PROGRAM BasketBadCtrl
VAR
	ARfbStnBadAssignCtrl: ARRAY [1..iStnQty] OF fbAssignBadBstCtrl;
	ARfbArmBadAssignCtrl: ARRAY [1..iArmQty] OF fbAssignBadBstCtrl;
	bGeneralAssignBadBasket: BOOL;

END_VAR

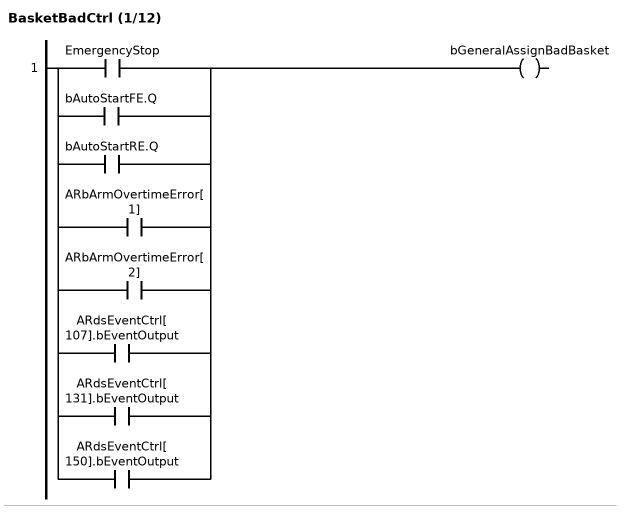
// NETWORK 1
bGeneralAssignBadBasket := EmergencyStop OR bAutoStartFE.Q OR bAutoStartRE.Q OR ARbArmOvertimeError[1] OR ARbArmOvertimeError[2] OR ARdsEventCtrl[107].bEventOutput OR ARdsEventCtrl[131].bEventOutput OR ARdsEventCtrl[150].bEventOutput;

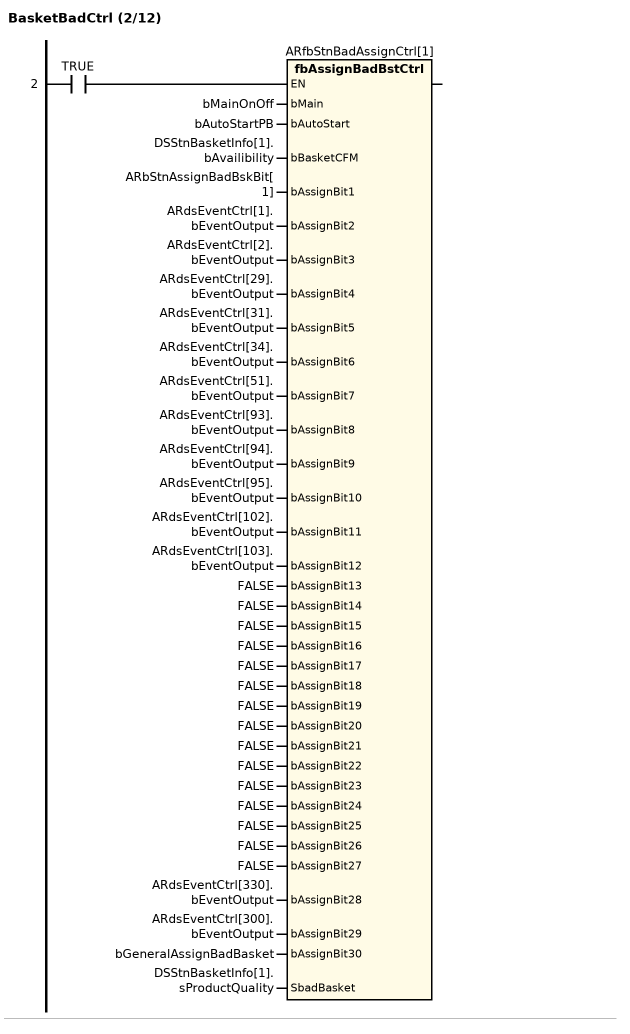
// NETWORK 2
ARfbStnBadAssignCtrl[1](
    bMain := bMainOnOff,
    bAutoStart := bAutoStartPB,
    bBasketCFM := DSStnBasketInfo[1].bAvailibility,
    bAssignBit1 := ARbStnAssignBadBskBit[1],
    bAssignBit2 := ARdsEventCtrl[1].bEventOutput,
    bAssignBit3 := ARdsEventCtrl[2].bEventOutput,
    bAssignBit4 := ARdsEventCtrl[29].bEventOutput,
    bAssignBit5 := ARdsEventCtrl[31].bEventOutput,
    bAssignBit6 := ARdsEventCtrl[34].bEventOutput,
    bAssignBit7 := ARdsEventCtrl[51].bEventOutput,
    bAssignBit8 := ARdsEventCtrl[93].bEventOutput,
    bAssignBit9 := ARdsEventCtrl[94].bEventOutput,
    bAssignBit10 := ARdsEventCtrl[95].bEventOutput,
    bAssignBit11 := ARdsEventCtrl[102].bEventOutput,
    bAssignBit12 := ARdsEventCtrl[103].bEventOutput,
    bAssignBit13 := FALSE,
    bAssignBit14 := FALSE,
    bAssignBit15 := FALSE,
    bAssignBit16 := FALSE,
    bAssignBit17 := FALSE,
    bAssignBit18 := FALSE,
    bAssignBit19 := FALSE,
    bAssignBit20 := FALSE,
    bAssignBit21 := FALSE,
    bAssignBit22 := FALSE,
    bAssignBit23 := FALSE,
    bAssignBit24 := FALSE,
    bAssignBit25 := FALSE,
    bAssignBit26 := FALSE,
    bAssignBit27 := FALSE,
    bAssignBit28 := ARdsEventCtrl[330].bEventOutput,
    bAssignBit29 := ARdsEventCtrl[300].bEventOutput,
    bAssignBit30 := bGeneralAssignBadBasket,
    SbadBasket := DSStnBasketInfo[1].sProductQuality); // fbAssignBadBstCtrl

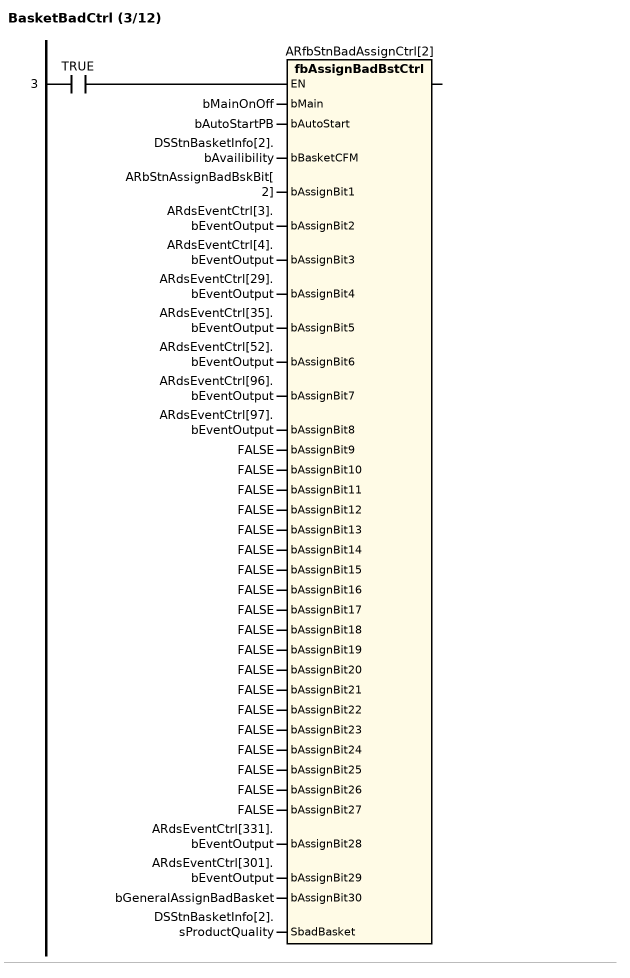
// NETWORK 3
ARfbStnBadAssignCtrl[2](
    bMain := bMainOnOff,
    bAutoStart := bAutoStartPB,
    bBasketCFM := DSStnBasketInfo[2].bAvailibility,
    bAssignBit1 := ARbStnAssignBadBskBit[2],
    bAssignBit2 := ARdsEventCtrl[3].bEventOutput,
    bAssignBit3 := ARdsEventCtrl[4].bEventOutput,
    bAssignBit4 := ARdsEventCtrl[29].bEventOutput,
    bAssignBit5 := ARdsEventCtrl[35].bEventOutput,
    bAssignBit6 := ARdsEventCtrl[52].bEventOutput,
    bAssignBit7 := ARdsEventCtrl[96].bEventOutput,
    bAssignBit8 := ARdsEventCtrl[97].bEventOutput,
    bAssignBit9 := FALSE,
    bAssignBit10 := FALSE,
    bAssignBit11 := FALSE,
    bAssignBit12 := FALSE,
    bAssignBit13 := FALSE,
    bAssignBit14 := FALSE,
    bAssignBit15 := FALSE,
    bAssignBit16 := FALSE,
    bAssignBit17 := FALSE,
    bAssignBit18 := FALSE,
    bAssignBit19 := FALSE,
    bAssignBit20 := FALSE,
    bAssignBit21 := FALSE,
    bAssignBit22 := FALSE,
    bAssignBit23 := FALSE,
    bAssignBit24 := FALSE,
    bAssignBit25 := FALSE,
    bAssignBit26 := FALSE,
    bAssignBit27 := FALSE,
    bAssignBit28 := ARdsEventCtrl[331].bEventOutput,
    bAssignBit29 := ARdsEventCtrl[301].bEventOutput,
    bAssignBit30 := bGeneralAssignBadBasket,
    SbadBasket := DSStnBasketInfo[2].sProductQuality); // fbAssignBadBstCtrl

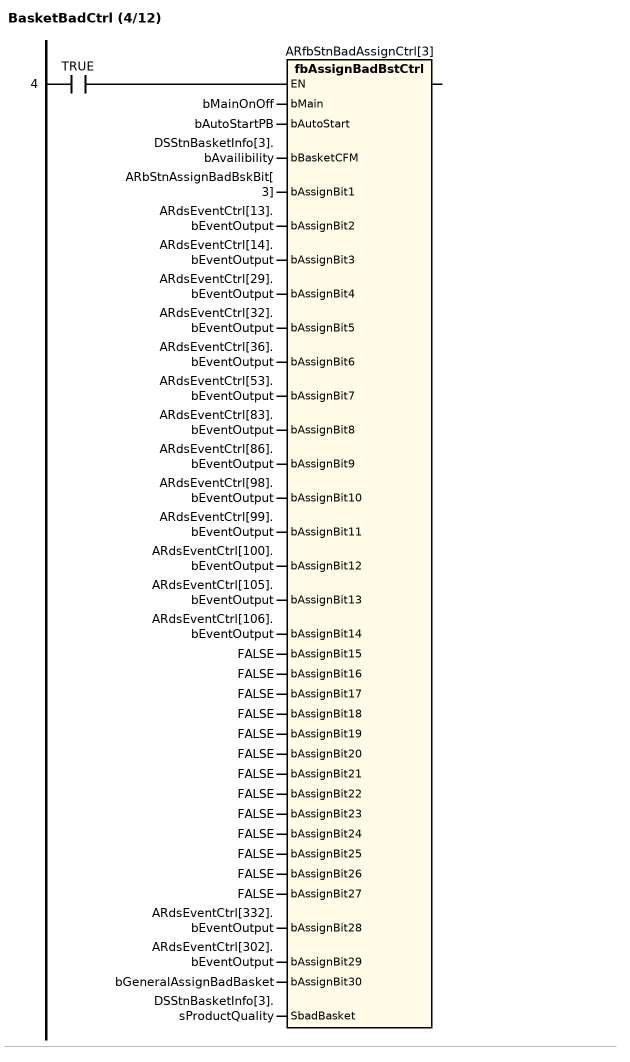
// NETWORK 4
ARfbStnBadAssignCtrl[3](
    bMain := bMainOnOff,
    bAutoStart := bAutoStartPB,
    bBasketCFM := DSStnBasketInfo[3].bAvailibility,
    bAssignBit1 := ARbStnAssignBadBskBit[3],
    bAssignBit2 := ARdsEventCtrl[13].bEventOutput,
    bAssignBit3 := ARdsEventCtrl[14].bEventOutput,
    bAssignBit4 := ARdsEventCtrl[29].bEventOutput,
    bAssignBit5 := ARdsEventCtrl[32].bEventOutput,
    bAssignBit6 := ARdsEventCtrl[36].bEventOutput,
    bAssignBit7 := ARdsEventCtrl[53].bEventOutput,
    bAssignBit8 := ARdsEventCtrl[83].bEventOutput,
    bAssignBit9 := ARdsEventCtrl[86].bEventOutput,
    bAssignBit10 := ARdsEventCtrl[98].bEventOutput,
    bAssignBit11 := ARdsEventCtrl[99].bEventOutput,
    bAssignBit12 := ARdsEventCtrl[100].bEventOutput,
    bAssignBit13 := ARdsEventCtrl[105].bEventOutput,
    bAssignBit14 := ARdsEventCtrl[106].bEventOutput,
    bAssignBit15 := FALSE,
    bAssignBit16 := FALSE,
    bAssignBit17 := FALSE,
    bAssignBit18 := FALSE,
    bAssignBit19 := FALSE,
    bAssignBit20 := FALSE,
    bAssignBit21 := FALSE,
    bAssignBit22 := FALSE,
    bAssignBit23 := FALSE,
    bAssignBit24 := FALSE,
    bAssignBit25 := FALSE,
    bAssignBit26 := FALSE,
    bAssignBit27 := FALSE,
    bAssignBit28 := ARdsEventCtrl[332].bEventOutput,
    bAssignBit29 := ARdsEventCtrl[302].bEventOutput,
    bAssignBit30 := bGeneralAssignBadBasket,
    SbadBasket := DSStnBasketInfo[3].sProductQuality); // fbAssignBadBstCtrl

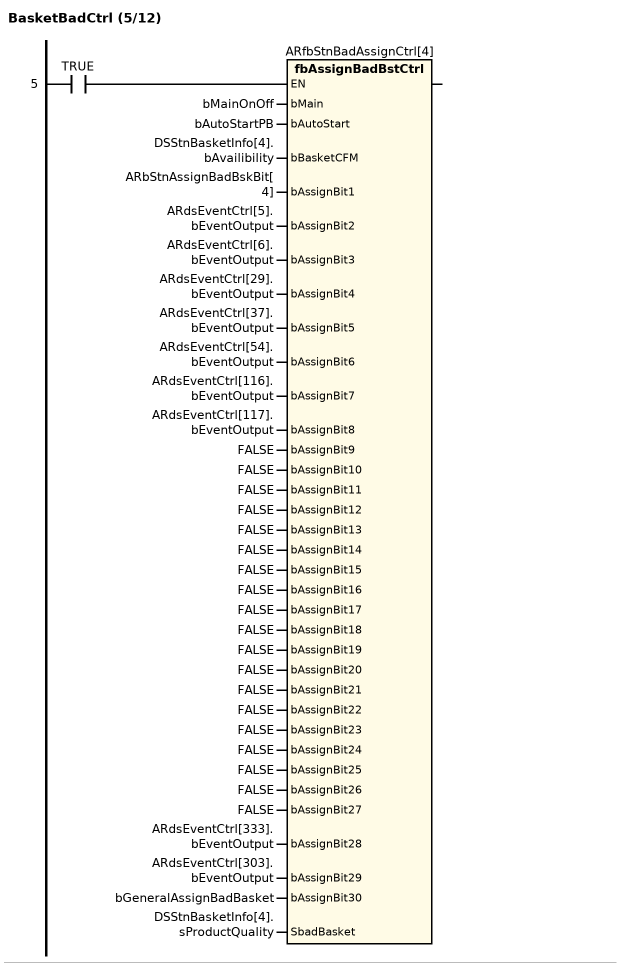
// NETWORK 5
ARfbStnBadAssignCtrl[4](
    bMain := bMainOnOff,
    bAutoStart := bAutoStartPB,
    bBasketCFM := DSStnBasketInfo[4].bAvailibility,
    bAssignBit1 := ARbStnAssignBadBskBit[4],
    bAssignBit2 := ARdsEventCtrl[5].bEventOutput,
    bAssignBit3 := ARdsEventCtrl[6].bEventOutput,
    bAssignBit4 := ARdsEventCtrl[29].bEventOutput,
    bAssignBit5 := ARdsEventCtrl[37].bEventOutput,
    bAssignBit6 := ARdsEventCtrl[54].bEventOutput,
    bAssignBit7 := ARdsEventCtrl[116].bEventOutput,
    bAssignBit8 := ARdsEventCtrl[117].bEventOutput,
    bAssignBit9 := FALSE,
    bAssignBit10 := FALSE,
    bAssignBit11 := FALSE,
    bAssignBit12 := FALSE,
    bAssignBit13 := FALSE,
    bAssignBit14 := FALSE,
    bAssignBit15 := FALSE,
    bAssignBit16 := FALSE,
    bAssignBit17 := FALSE,
    bAssignBit18 := FALSE,
    bAssignBit19 := FALSE,
    bAssignBit20 := FALSE,
    bAssignBit21 := FALSE,
    bAssignBit22 := FALSE,
    bAssignBit23 := FALSE,
    bAssignBit24 := FALSE,
    bAssignBit25 := FALSE,
    bAssignBit26 := FALSE,
    bAssignBit27 := FALSE,
    bAssignBit28 := ARdsEventCtrl[333].bEventOutput,
    bAssignBit29 := ARdsEventCtrl[303].bEventOutput,
    bAssignBit30 := bGeneralAssignBadBasket,
    SbadBasket := DSStnBasketInfo[4].sProductQuality); // fbAssignBadBstCtrl

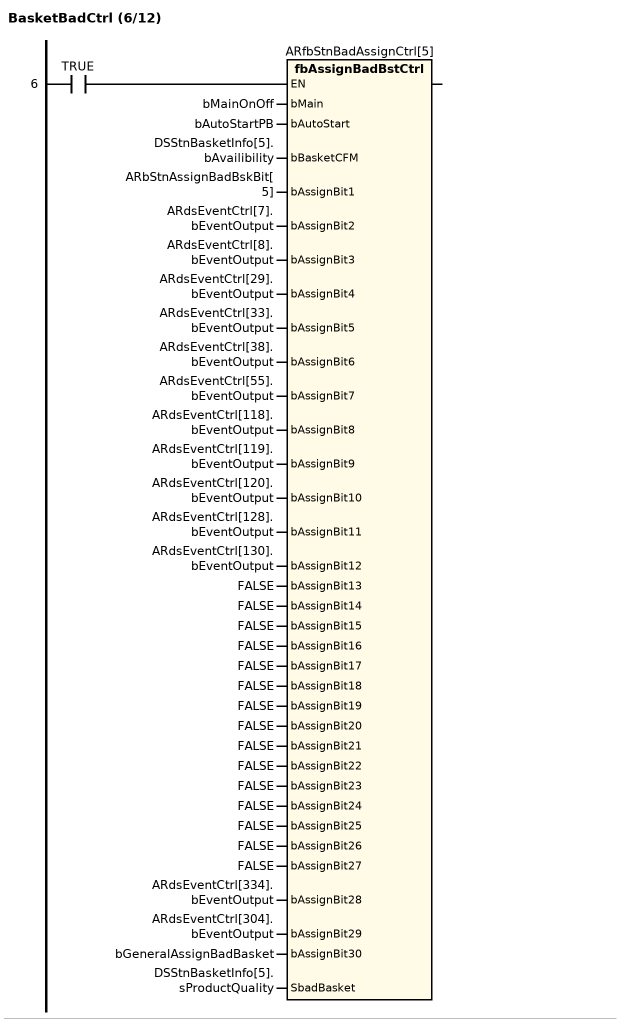
// NETWORK 6
ARfbStnBadAssignCtrl[5](
    bMain := bMainOnOff,
    bAutoStart := bAutoStartPB,
    bBasketCFM := DSStnBasketInfo[5].bAvailibility,
    bAssignBit1 := ARbStnAssignBadBskBit[5],
    bAssignBit2 := ARdsEventCtrl[7].bEventOutput,
    bAssignBit3 := ARdsEventCtrl[8].bEventOutput,
    bAssignBit4 := ARdsEventCtrl[29].bEventOutput,
    bAssignBit5 := ARdsEventCtrl[33].bEventOutput,
    bAssignBit6 := ARdsEventCtrl[38].bEventOutput,
    bAssignBit7 := ARdsEventCtrl[55].bEventOutput,
    bAssignBit8 := ARdsEventCtrl[118].bEventOutput,
    bAssignBit9 := ARdsEventCtrl[119].bEventOutput,
    bAssignBit10 := ARdsEventCtrl[120].bEventOutput,
    bAssignBit11 := ARdsEventCtrl[128].bEventOutput,
    bAssignBit12 := ARdsEventCtrl[130].bEventOutput,
    bAssignBit13 := FALSE,
    bAssignBit14 := FALSE,
    bAssignBit15 := FALSE,
    bAssignBit16 := FALSE,
    bAssignBit17 := FALSE,
    bAssignBit18 := FALSE,
    bAssignBit19 := FALSE,
    bAssignBit20 := FALSE,
    bAssignBit21 := FALSE,
    bAssignBit22 := FALSE,
    bAssignBit23 := FALSE,
    bAssignBit24 := FALSE,
    bAssignBit25 := FALSE,
    bAssignBit26 := FALSE,
    bAssignBit27 := FALSE,
    bAssignBit28 := ARdsEventCtrl[334].bEventOutput,
    bAssignBit29 := ARdsEventCtrl[304].bEventOutput,
    bAssignBit30 := bGeneralAssignBadBasket,
    SbadBasket := DSStnBasketInfo[5].sProductQuality); // fbAssignBadBstCtrl

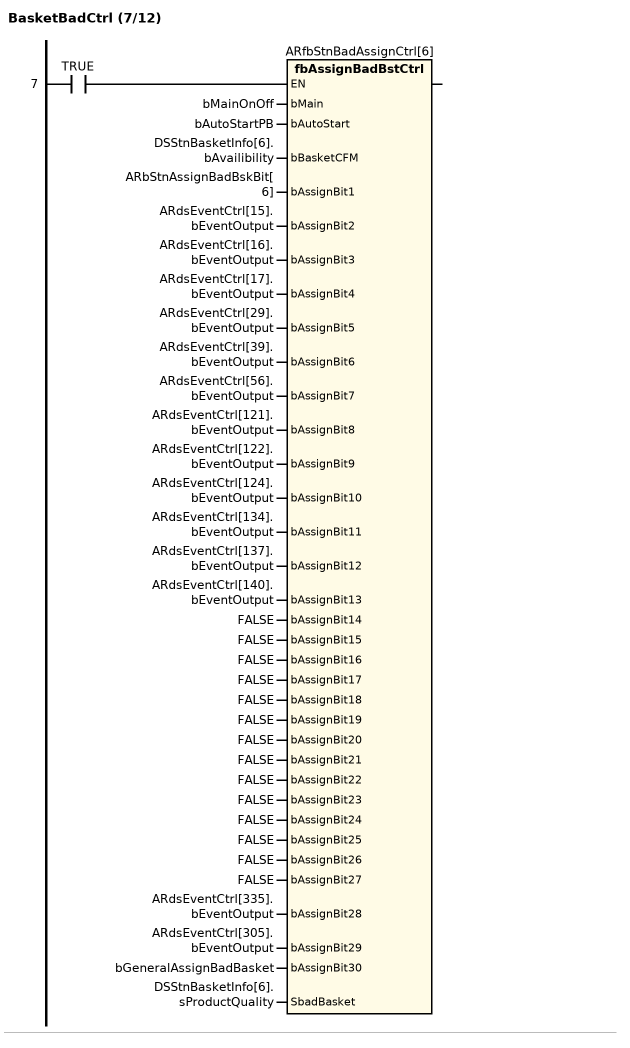
// NETWORK 7
ARfbStnBadAssignCtrl[6](
    bMain := bMainOnOff,
    bAutoStart := bAutoStartPB,
    bBasketCFM := DSStnBasketInfo[6].bAvailibility,
    bAssignBit1 := ARbStnAssignBadBskBit[6],
    bAssignBit2 := ARdsEventCtrl[15].bEventOutput,
    bAssignBit3 := ARdsEventCtrl[16].bEventOutput,
    bAssignBit4 := ARdsEventCtrl[17].bEventOutput,
    bAssignBit5 := ARdsEventCtrl[29].bEventOutput,
    bAssignBit6 := ARdsEventCtrl[39].bEventOutput,
    bAssignBit7 := ARdsEventCtrl[56].bEventOutput,
    bAssignBit8 := ARdsEventCtrl[121].bEventOutput,
    bAssignBit9 := ARdsEventCtrl[122].bEventOutput,
    bAssignBit10 := ARdsEventCtrl[124].bEventOutput,
    bAssignBit11 := ARdsEventCtrl[134].bEventOutput,
    bAssignBit12 := ARdsEventCtrl[137].bEventOutput,
    bAssignBit13 := ARdsEventCtrl[140].bEventOutput,
    bAssignBit14 := FALSE,
    bAssignBit15 := FALSE,
    bAssignBit16 := FALSE,
    bAssignBit17 := FALSE,
    bAssignBit18 := FALSE,
    bAssignBit19 := FALSE,
    bAssignBit20 := FALSE,
    bAssignBit21 := FALSE,
    bAssignBit22 := FALSE,
    bAssignBit23 := FALSE,
    bAssignBit24 := FALSE,
    bAssignBit25 := FALSE,
    bAssignBit26 := FALSE,
    bAssignBit27 := FALSE,
    bAssignBit28 := ARdsEventCtrl[335].bEventOutput,
    bAssignBit29 := ARdsEventCtrl[305].bEventOutput,
    bAssignBit30 := bGeneralAssignBadBasket,
    SbadBasket := DSStnBasketInfo[6].sProductQuality); // fbAssignBadBstCtrl

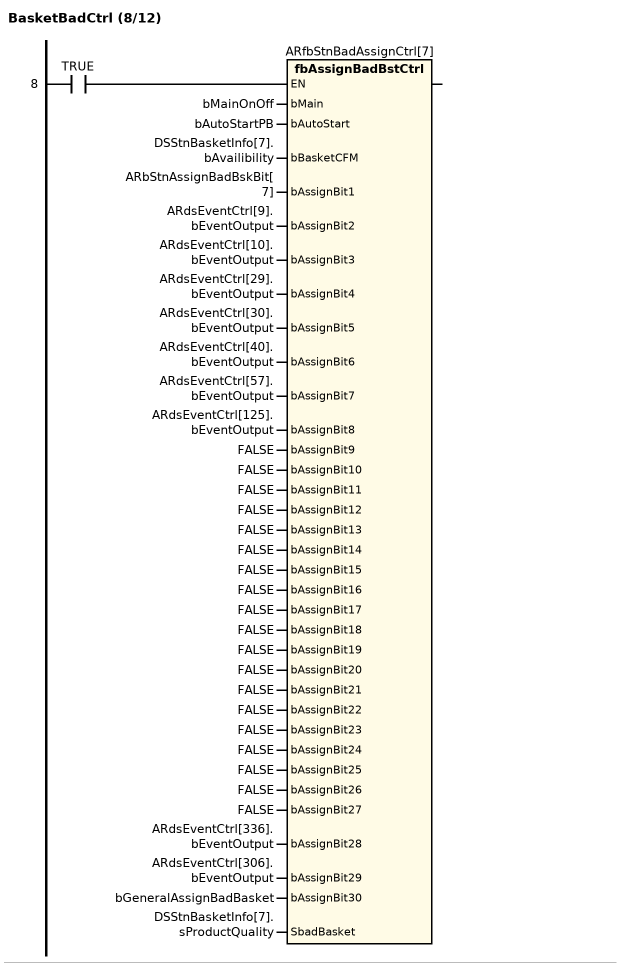
// NETWORK 8
ARfbStnBadAssignCtrl[7](
    bMain := bMainOnOff,
    bAutoStart := bAutoStartPB,
    bBasketCFM := DSStnBasketInfo[7].bAvailibility,
    bAssignBit1 := ARbStnAssignBadBskBit[7],
    bAssignBit2 := ARdsEventCtrl[9].bEventOutput,
    bAssignBit3 := ARdsEventCtrl[10].bEventOutput,
    bAssignBit4 := ARdsEventCtrl[29].bEventOutput,
    bAssignBit5 := ARdsEventCtrl[30].bEventOutput,
    bAssignBit6 := ARdsEventCtrl[40].bEventOutput,
    bAssignBit7 := ARdsEventCtrl[57].bEventOutput,
    bAssignBit8 := ARdsEventCtrl[125].bEventOutput,
    bAssignBit9 := FALSE,
    bAssignBit10 := FALSE,
    bAssignBit11 := FALSE,
    bAssignBit12 := FALSE,
    bAssignBit13 := FALSE,
    bAssignBit14 := FALSE,
    bAssignBit15 := FALSE,
    bAssignBit16 := FALSE,
    bAssignBit17 := FALSE,
    bAssignBit18 := FALSE,
    bAssignBit19 := FALSE,
    bAssignBit20 := FALSE,
    bAssignBit21 := FALSE,
    bAssignBit22 := FALSE,
    bAssignBit23 := FALSE,
    bAssignBit24 := FALSE,
    bAssignBit25 := FALSE,
    bAssignBit26 := FALSE,
    bAssignBit27 := FALSE,
    bAssignBit28 := ARdsEventCtrl[336].bEventOutput,
    bAssignBit29 := ARdsEventCtrl[306].bEventOutput,
    bAssignBit30 := bGeneralAssignBadBasket,
    SbadBasket := DSStnBasketInfo[7].sProductQuality); // fbAssignBadBstCtrl

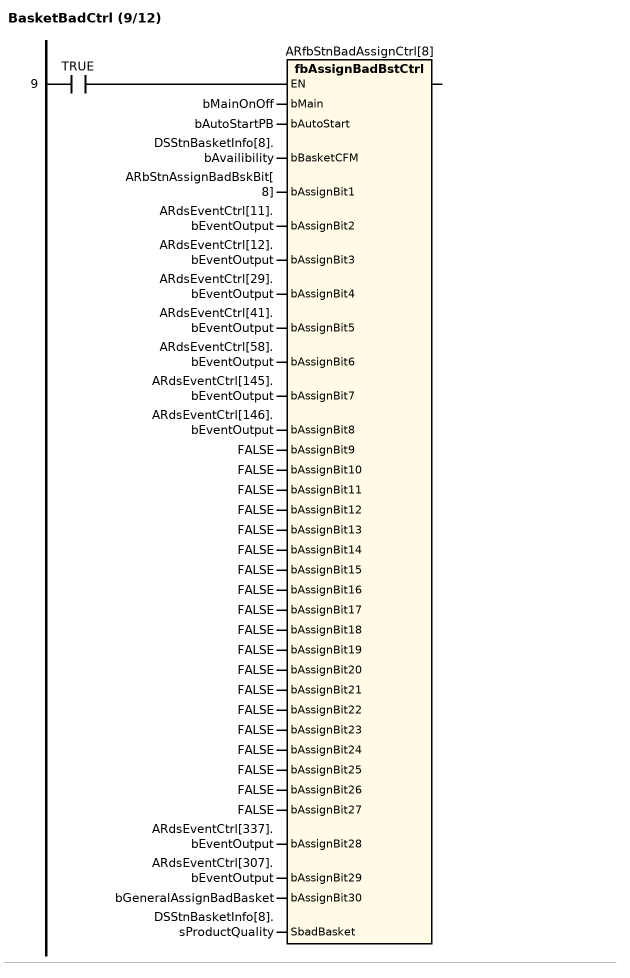
// NETWORK 9
ARfbStnBadAssignCtrl[8](
    bMain := bMainOnOff,
    bAutoStart := bAutoStartPB,
    bBasketCFM := DSStnBasketInfo[8].bAvailibility,
    bAssignBit1 := ARbStnAssignBadBskBit[8],
    bAssignBit2 := ARdsEventCtrl[11].bEventOutput,
    bAssignBit3 := ARdsEventCtrl[12].bEventOutput,
    bAssignBit4 := ARdsEventCtrl[29].bEventOutput,
    bAssignBit5 := ARdsEventCtrl[41].bEventOutput,
    bAssignBit6 := ARdsEventCtrl[58].bEventOutput,
    bAssignBit7 := ARdsEventCtrl[145].bEventOutput,
    bAssignBit8 := ARdsEventCtrl[146].bEventOutput,
    bAssignBit9 := FALSE,
    bAssignBit10 := FALSE,
    bAssignBit11 := FALSE,
    bAssignBit12 := FALSE,
    bAssignBit13 := FALSE,
    bAssignBit14 := FALSE,
    bAssignBit15 := FALSE,
    bAssignBit16 := FALSE,
    bAssignBit17 := FALSE,
    bAssignBit18 := FALSE,
    bAssignBit19 := FALSE,
    bAssignBit20 := FALSE,
    bAssignBit21 := FALSE,
    bAssignBit22 := FALSE,
    bAssignBit23 := FALSE,
    bAssignBit24 := FALSE,
    bAssignBit25 := FALSE,
    bAssignBit26 := FALSE,
    bAssignBit27 := FALSE,
    bAssignBit28 := ARdsEventCtrl[337].bEventOutput,
    bAssignBit29 := ARdsEventCtrl[307].bEventOutput,
    bAssignBit30 := bGeneralAssignBadBasket,
    SbadBasket := DSStnBasketInfo[8].sProductQuality); // fbAssignBadBstCtrl

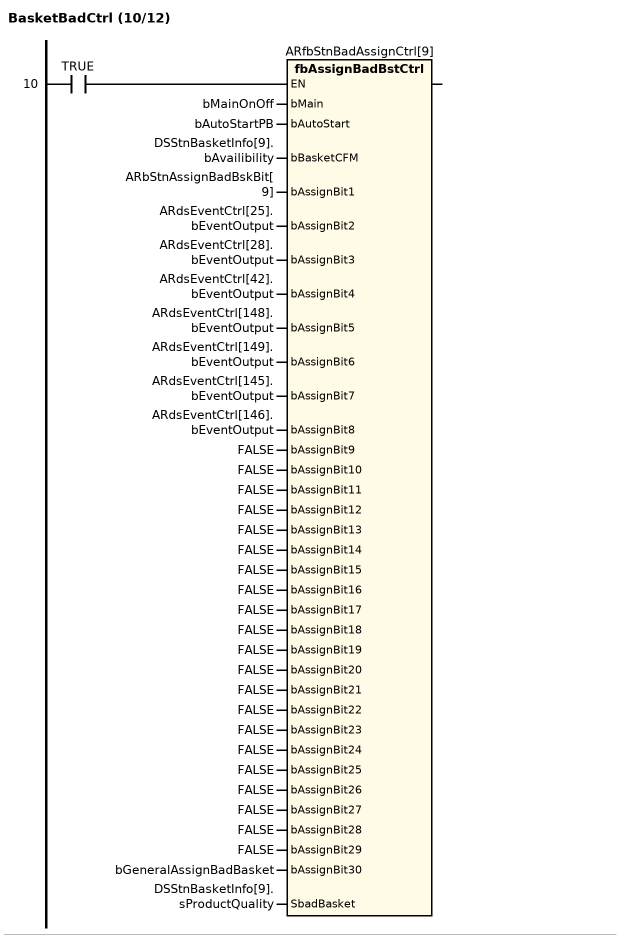
// NETWORK 10
ARfbStnBadAssignCtrl[9](
    bMain := bMainOnOff,
    bAutoStart := bAutoStartPB,
    bBasketCFM := DSStnBasketInfo[9].bAvailibility,
    bAssignBit1 := ARbStnAssignBadBskBit[9],
    bAssignBit2 := ARdsEventCtrl[25].bEventOutput,
    bAssignBit3 := ARdsEventCtrl[28].bEventOutput,
    bAssignBit4 := ARdsEventCtrl[42].bEventOutput,
    bAssignBit5 := ARdsEventCtrl[148].bEventOutput,
    bAssignBit6 := ARdsEventCtrl[149].bEventOutput,
    bAssignBit7 := ARdsEventCtrl[145].bEventOutput,
    bAssignBit8 := ARdsEventCtrl[146].bEventOutput,
    bAssignBit9 := FALSE,
    bAssignBit10 := FALSE,
    bAssignBit11 := FALSE,
    bAssignBit12 := FALSE,
    bAssignBit13 := FALSE,
    bAssignBit14 := FALSE,
    bAssignBit15 := FALSE,
    bAssignBit16 := FALSE,
    bAssignBit17 := FALSE,
    bAssignBit18 := FALSE,
    bAssignBit19 := FALSE,
    bAssignBit20 := FALSE,
    bAssignBit21 := FALSE,
    bAssignBit22 := FALSE,
    bAssignBit23 := FALSE,
    bAssignBit24 := FALSE,
    bAssignBit25 := FALSE,
    bAssignBit26 := FALSE,
    bAssignBit27 := FALSE,
    bAssignBit28 := FALSE,
    bAssignBit29 := FALSE,
    bAssignBit30 := bGeneralAssignBadBasket,
    SbadBasket := DSStnBasketInfo[9].sProductQuality); // fbAssignBadBstCtrl

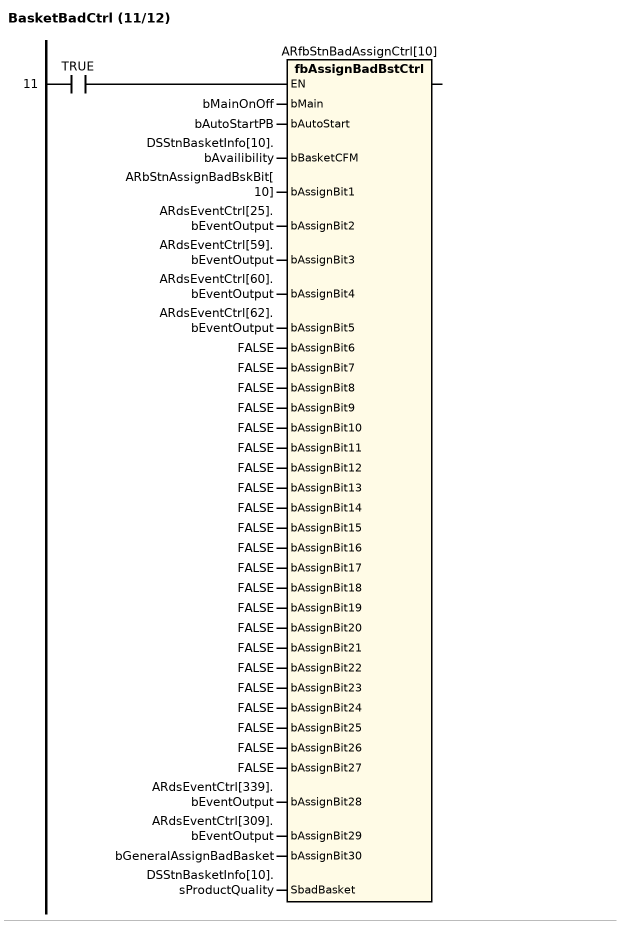
// NETWORK 11
ARfbStnBadAssignCtrl[10](
    bMain := bMainOnOff,
    bAutoStart := bAutoStartPB,
    bBasketCFM := DSStnBasketInfo[10].bAvailibility,
    bAssignBit1 := ARbStnAssignBadBskBit[10],
    bAssignBit2 := ARdsEventCtrl[25].bEventOutput,
    bAssignBit3 := ARdsEventCtrl[59].bEventOutput,
    bAssignBit4 := ARdsEventCtrl[60].bEventOutput,
    bAssignBit5 := ARdsEventCtrl[62].bEventOutput,
    bAssignBit6 := FALSE,
    bAssignBit7 := FALSE,
    bAssignBit8 := FALSE,
    bAssignBit9 := FALSE,
    bAssignBit10 := FALSE,
    bAssignBit11 := FALSE,
    bAssignBit12 := FALSE,
    bAssignBit13 := FALSE,
    bAssignBit14 := FALSE,
    bAssignBit15 := FALSE,
    bAssignBit16 := FALSE,
    bAssignBit17 := FALSE,
    bAssignBit18 := FALSE,
    bAssignBit19 := FALSE,
    bAssignBit20 := FALSE,
    bAssignBit21 := FALSE,
    bAssignBit22 := FALSE,
    bAssignBit23 := FALSE,
    bAssignBit24 := FALSE,
    bAssignBit25 := FALSE,
    bAssignBit26 := FALSE,
    bAssignBit27 := FALSE,
    bAssignBit28 := ARdsEventCtrl[339].bEventOutput,
    bAssignBit29 := ARdsEventCtrl[309].bEventOutput,
    bAssignBit30 := bGeneralAssignBadBasket,
    SbadBasket := DSStnBasketInfo[10].sProductQuality); // fbAssignBadBstCtrl

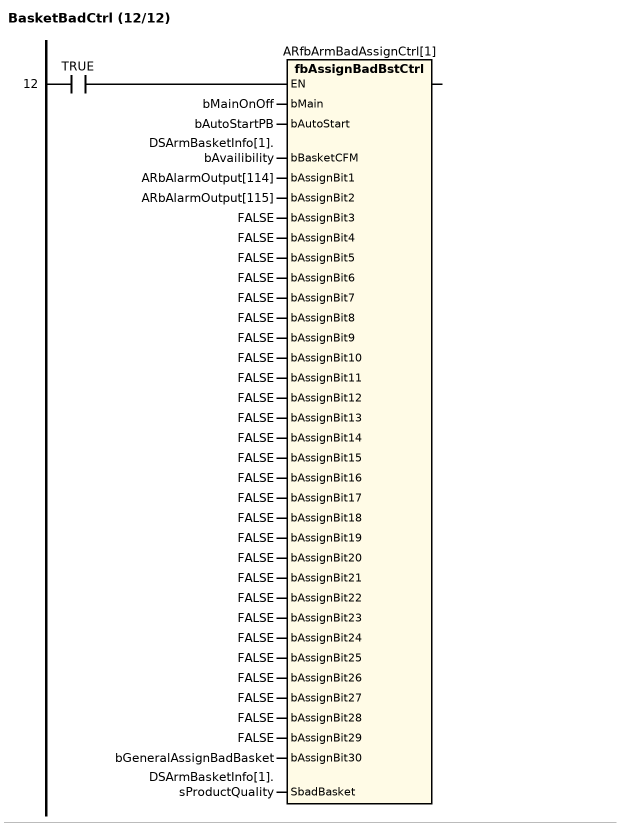
// NETWORK 12
ARfbArmBadAssignCtrl[1](
    bMain := bMainOnOff,
    bAutoStart := bAutoStartPB,
    bBasketCFM := DSArmBasketInfo[1].bAvailibility,
    bAssignBit1 := ARbAlarmOutput[114],
    bAssignBit2 := ARbAlarmOutput[115],
    bAssignBit3 := FALSE,
    bAssignBit4 := FALSE,
    bAssignBit5 := FALSE,
    bAssignBit6 := FALSE,
    bAssignBit7 := FALSE,
    bAssignBit8 := FALSE,
    bAssignBit9 := FALSE,
    bAssignBit10 := FALSE,
    bAssignBit11 := FALSE,
    bAssignBit12 := FALSE,
    bAssignBit13 := FALSE,
    bAssignBit14 := FALSE,
    bAssignBit15 := FALSE,
    bAssignBit16 := FALSE,
    bAssignBit17 := FALSE,
    bAssignBit18 := FALSE,
    bAssignBit19 := FALSE,
    bAssignBit20 := FALSE,
    bAssignBit21 := FALSE,
    bAssignBit22 := FALSE,
    bAssignBit23 := FALSE,
    bAssignBit24 := FALSE,
    bAssignBit25 := FALSE,
    bAssignBit26 := FALSE,
    bAssignBit27 := FALSE,
    bAssignBit28 := FALSE,
    bAssignBit29 := FALSE,
    bAssignBit30 := bGeneralAssignBadBasket,
    SbadBasket := DSArmBasketInfo[1].sProductQuality); // fbAssignBadBstCtrl

END_PROGRAM

(* stored: Version 1.1.0.1, ProductVersion 3.1.4024.12
   POU BasketBadCtrl: Id {b6e47355-c24f-4b8d-a565-89587770cbac}, SpecialFunc None *)
